    W =  -179.868 deg,    P =   -0.088 deg,    R =   -0.987 deg
};
P[363]{
   GP1:
    UF : 0, UT : 6,      CONFIG : 'N U T, 0, 0, 0',
    X =  350011.060  mm,    Y =   38.933  mm,    Z =   -325807.670  mm,
    W =  -179.992 deg,    P =   0.026 deg,    R =   -1.000 deg
};
P[364]{
   GP1:
    UF : 0, UT : 6,      CONFIG : 'N U T, 0, 0, 0',
    X =  350006.343  mm,    Y =   43.364  mm,    Z =   -325807.400  mm,
    W =  -179.999 deg,    P =   0.015 deg,    R =   -1.000 deg
};
P[365]{
   GP1:
    UF : 0, UT : 6,      CONFIG : 'N U T, 0, 0, 0',
    X =  349940.173  mm,    Y =   106.113  mm,    Z =   -325807.458  mm,
    W =  -179.846 deg,    P =   -0.075 deg,    R =   -0.985 deg
};
P[366]{
   GP1:
    UF : 0, UT : 6,      CONFIG : 'N U T, 0, 0, 0',
    X =  350114.721  mm,    Y =   -100.490  mm,    Z =   -325807.810  mm,
    W =  -180.070 deg,    P =   -0.016 deg,    R =   -0.997 deg
};
P[367]{
   GP1:
    UF : 0, UT : 6,      CONFIG : 'N U T, 0, 0, 0',
    X =  350023.392  mm,    Y =   -22.593  mm,    Z =   -325807.668  mm,
    W =  -179.928 deg,    P =   0.086 deg,    R =   -0.994 deg
};
P[368]{
   GP1:
    UF : 0, UT : 6,      CONFIG : 'N U T, 0, 0, 0',
    X =  349970.490  mm,    Y =   8.398  mm,    Z =   -325807.460  mm,
    W =  -180.011 deg,    P =   0.065 deg,    R =   -0.998 deg
};
P[369]{
   GP1:
    UF : 0, UT : 6,      CONFIG : 'N U T, 0, 0, 0',
    X =  349963.107  mm,    Y =   15.166  mm,    Z =   -325807.480  mm,
    W =  -180.007 deg,    P =   0.054 deg,    R =   -0.999 deg
};
P[370]{
   GP1:
    UF : 0, UT : 6,      CONFIG : 'N U T, 0, 0, 0',
    X =  349967.577  mm,    Y =   4.673  mm,    Z =   -325807.453  mm,
    W =  -180.013 deg,    P =   0.068 deg,    R =   -0.998 deg
};
P[371]{
   GP1:
    UF : 0, UT : 6,      CONFIG : 'N U T, 0, 0, 0',
    X =  349899.498  mm,    Y =   72.748  mm,    Z =   -325807.453  mm,
    W =  -179.870 deg,    P =   0.045 deg,    R =   -0.990 deg
};
P[372]{
   GP1:
    UF : 0, UT : 6,      CONFIG : 'N U T, 0, 0, 0',
    X =  349940.962  mm,    Y =   6.715  mm,    Z =   -325807.602  mm,
    W =  -180.025 deg,    P =   0.099 deg,    R =   -0.995 deg
};
P[373]{
   GP1:
    UF : 0, UT : 6,      CONFIG : 'N U T, 0, 0, 0',
    X =  349988.685  mm,    Y =   -47.181  mm,    Z =   -325807.339  mm,
    W =  -179.937 deg,    P =   0.123 deg,    R =   -0.990 deg
};
P[374]{
   GP1:
    UF : 0, UT : 6,      CONFIG : 'N U T, 0, 0, 0',
    X =  349935.723  mm,    Y =   5.743  mm,    Z =   -325807.701  mm,
    W =  -180.019 deg,    P =   0.118 deg,    R =   -0.993 deg
};
P[375]{
   GP1:
    UF : 0, UT : 6,      CONFIG : 'N U T, 0, 0, 0',
    X =  350040.680  mm,    Y =   -104.256  mm,    Z =   -325807.539  mm,
    W =  -179.944 deg,    P =   0.142 deg,    R =   -0.988 deg
};
P[376]{
   GP1:
    UF : 0, UT : 6,      CONFIG : 'N U T, 0, 0, 0',
    X =  349988.847  mm,    Y =   -58.050  mm,    Z =   -325808.015  mm,
    W =  -179.918 deg,    P =   0.146 deg,    R =   -0.986 deg
};
P[377]{
   GP1:
    UF : 0, UT : 6,      CONFIG : 'N U T, 0, 0, 0',
    X =  350008.350  mm,    Y =   -81.087  mm,    Z =   -325807.613  mm,
    W =  -179.907 deg,    P =   0.202 deg,    R =   -0.975 deg
};
P[378]{
   GP1:
    UF : 0, UT : 6,      CONFIG : 'N U T, 0, 0, 0',
    X =  349912.927  mm,    Y =   4.381  mm,    Z =   -325807.326  mm,
    W =  -180.014 deg,    P =   0.201 deg,    R =   -0.979 deg
};
P[379]{
   GP1:
    UF : 0, UT : 6,      CONFIG : 'N U T, 0, 0, 0',
    X =  349880.747  mm,    Y =   35.030  mm,    Z =   -325807.873  mm,
    W =  -179.887 deg,    P =   0.143 deg,    R =   -0.983 deg
};
P[380]{
   GP1:
    UF : 0, UT : 6,      CONFIG : 'N U T, 0, 0, 0',
    X =  349881.008  mm,    Y =   17.753  mm,    Z =   -325807.522  mm,
    W =  -179.929 deg,    P =   0.180 deg,    R =   -0.981 deg
};
P[381]{
   GP1:
    UF : 0, UT : 6,      CONFIG : 'N U T, 0, 0, 0',
    X =  350037.899  mm,    Y =   6.412  mm,    Z =   -325808.221  mm,
    W =  -179.934 deg,    P =   0.055 deg,    R =   -0.996 deg
};
P[382]{
   GP1:
    UF : 0, UT : 6,      CONFIG : 'N U T, 0, 0, 0',
    X =  350031.037  mm,    Y =   12.249  mm,    Z =   -325808.736  mm,
    W =  -179.955 deg,    P =   0.053 deg,    R =   -0.998 deg
};
P[383]{
   GP1:
    UF : 0, UT : 6,      CONFIG : 'N U T, 0, 0, 0',
    X =  349899.914  mm,    Y =   79.737  mm,    Z =   -325808.810  mm,
    W =  -179.855 deg,    P =   0.036 deg,    R =   -0.989 deg
};
P[384]{
   GP1:
    UF : 0, UT : 6,      CONFIG : 'N U T, 0, 0, 0',
    X =  349969.792  mm,    Y =   1.424  mm,    Z =   -325808.974  mm,
    W =  -180.009 deg,    P =   0.069 deg,    R =   -0.998 deg
};
P[385]{
   GP1:
    UF : 0, UT : 6,      CONFIG : 'N U T, 0, 0, 0',
    X =  349960.411  mm,    Y =   10.805  mm,    Z =   -325808.974  mm,
    W =  -180.014 deg,    P =   0.066 deg,    R =   -0.998 deg
};
P[386]{
   GP1:
    UF : 0, UT : 6,      CONFIG : 'N U T, 0, 0, 0',
    X =  349963.050  mm,    Y =   0.566  mm,    Z =   -325808.599  mm,
    W =  -180.017 deg,    P =   0.081 deg,    R =   -0.997 deg
};
P[387]{
   GP1:
    UF : 0, UT : 6,      CONFIG : 'N U T, 0, 0, 0',
    X =  349955.646  mm,    Y =   7.674  mm,    Z =   -325809.075  mm,
    W =  -180.018 deg,    P =   0.078 deg,    R =   -0.997 deg
};
P[388]{
   GP1:
    UF : 0, UT : 6,      CONFIG : 'N U T, 0, 0, 0',
    X =  349892.240  mm,    Y =   70.955  mm,    Z =   -325808.835  mm,
    W =  -179.851 deg,    P =   0.070 deg,    R =   -0.986 deg
};
P[389]{
   GP1:
    UF : 0, UT : 6,      CONFIG : 'N U T, 0, 0, 0',
    X =  349890.827  mm,    Y =   57.371  mm,    Z =   -325808.189  mm,
    W =  -179.868 deg,    P =   0.084 deg,    R =   -0.988 deg
};
P[390]{
   GP1:
    UF : 0, UT : 6,      CONFIG : 'N U T, 0, 0, 0',
    X =  349904.306  mm,    Y =   0.938  mm,    Z =   -325808.338  mm,
    W =  -180.017 deg,    P =   0.214 deg,    R =   -0.977 deg
};
P[391]{
   GP1:
    UF : 0, UT : 6,      CONFIG : 'N U T, 0, 0, 0',
    X =  349895.241  mm,    Y =   5.574  mm,    Z =   -325808.287  mm,
    W =  -180.000 deg,    P =   0.196 deg,    R =   -0.981 deg
};
P[392]{
   GP1:
    UF : 0, UT : 6,      CONFIG : 'N U T, 0, 0, 0',
    X =  350127.266  mm,    Y =   -37.191  mm,    Z =   -325809.968  mm,
    W =  -180.039 deg,    P =   -0.112 deg,    R =   -0.993 deg
};
P[393]{
   GP1:
    UF : 0, UT : 6,      CONFIG : 'N U T, 0, 0, 0',
    X =  349998.625  mm,    Y =   66.854  mm,    Z =   -325809.775  mm,
    W =  -180.004 deg,    P =   -0.072 deg,    R =   -0.997 deg
};
P[394]{
   GP1:
    UF : 0, UT : 6,      CONFIG : 'N U T, 0, 0, 0',
    X =  350025.040  mm,    Y =   19.677  mm,    Z =   -325809.276  mm,
    W =  -179.962 deg,    P =   0.065 deg,    R =   -0.997 deg
};
P[395]{
   GP1:
    UF : 0, UT : 6,      CONFIG : 'N U T, 0, 0, 0',
    X =  349931.313  mm,    Y =   110.110  mm,    Z =   -325809.292  mm,
    W =  -179.819 deg,    P =   -0.074 deg,    R =   -0.981 deg
};
P[396]{
   GP1:
    UF : 0, UT : 6,      CONFIG : 'N U T, 0, 0, 0',
    X =  349924.018  mm,    Y =   108.625  mm,    Z =   -325809.284  mm,
    W =  -179.816 deg,    P =   -0.057 deg,    R =   -0.981 deg
};
P[397]{
   GP1:
    UF : 0, UT : 6,      CONFIG : 'N U T, 0, 0, 0',
    X =  350035.241  mm,    Y =   -29.808  mm,    Z =   -325809.701  mm,
    W =  -179.920 deg,    P =   0.069 deg,    R =   -0.994 deg
};
P[398]{
   GP1:
    UF : 0, UT : 6,      CONFIG : 'N U T, 0, 0, 0',
    X =  349908.694  mm,    Y =   94.566  mm,    Z =   -325809.383  mm,
    W =  -179.840 deg,    P =   0.012 deg,    R =   -0.987 deg
};
P[399]{
   GP1:
    UF : 0, UT : 6,      CONFIG : 'N U T, 0, 0, 0',
    X =  350112.602  mm,    Y =   -111.159  mm,    Z =   -325810.070  mm,
    W =  -180.076 deg,    P =   -0.007 deg,    R =   -0.997 deg
};
P[400]{
   GP1:
    UF : 0, UT : 6,      CONFIG : 'N U T, 0, 0, 0',
    X =  350036.736  mm,    Y =   -53.058  mm,    Z =   -325809.103  mm,
    W =  -179.927 deg,    P =   0.076 deg,    R =   -0.994 deg
};
P[401]{
   GP1:
    UF : 0, UT : 6,      CONFIG : 'N U T, 0, 0, 0',
    X =  349893.364  mm,    Y =   76.907  mm,    Z =   -325809.706  mm,
    W =  -179.845 deg,    P =   0.053 deg,    R =   -0.986 deg
};
P[402]{
   GP1:
    UF : 0, UT : 6,      CONFIG : 'N U T, 0, 0, 0',
    X =  349997.088  mm,    Y =   -37.551  mm,    Z =   -325809.501  mm,
    W =  -179.936 deg,    P =   0.119 deg,    R =   -0.991 deg
};
P[403]{
   GP1:
    UF : 0, UT : 6,      CONFIG : 'N U T, 0, 0, 0',
    X =  349967.622  mm,    Y =   -7.327  mm,    Z =   -325809.623  mm,
    W =  -180.014 deg,    P =   0.082 deg,    R =   -0.997 deg
};
P[404]{
   GP1:
    UF : 0, UT : 6,      CONFIG : 'N U T, 0, 0, 0',
    X =  349990.888  mm,    Y =   -41.278  mm,    Z =   -325809.201  mm,
    W =  -179.938 deg,    P =   0.119 deg,    R =   -0.991 deg
};
P[405]{
   GP1:
    UF : 0, UT : 6,      CONFIG : 'N U T, 0, 0, 0',
    X =  349961.948  mm,    Y =   -13.770  mm,    Z =   -325809.419  mm,
    W =  -180.014 deg,    P =   0.096 deg,    R =   -0.995 deg
};
P[406]{
   GP1:
    UF : 0, UT : 6,      CONFIG : 'N U T, 0, 0, 0',
    X =  349954.785  mm,    Y =   -6.599  mm,    Z =   -325809.589  mm,
    W =  -180.024 deg,    P =   0.096 deg,    R =   -0.995 deg
};
P[407]{
   GP1:
    UF : 0, UT : 6,      CONFIG : 'N U T, 0, 0, 0',
    X =  349947.731  mm,    Y =   0.463  mm,    Z =   -325809.430  mm,
    W =  -180.027 deg,    P =   0.099 deg,    R =   -0.995 deg
};
P[408]{
   GP1:
    UF : 0, UT : 6,      CONFIG : 'N U T, 0, 0, 0',
    X =  349968.821  mm,    Y =   -21.469  mm,    Z =   -325809.248  mm,
    W =  -180.002 deg,    P =   0.095 deg,    R =   -0.995 deg
};
P[409]{
   GP1:
    UF : 0, UT : 6,      CONFIG : 'N U T, 0, 0, 0',
    X =  349982.592  mm,    Y =   -50.508  mm,    Z =   -325809.611  mm,
    W =  -179.939 deg,    P =   0.124 deg,    R =   -0.990 deg
};
P[410]{
   GP1:
    UF : 0, UT : 6,      CONFIG : 'N U T, 0, 0, 0',
    X =  349925.706  mm,    Y =   6.623  mm,    Z =   -325809.710  mm,
    W =  -180.017 deg,    P =   0.162 deg,    R =   -0.987 deg
};
P[411]{
   GP1:
    UF : 0, UT : 6,      CONFIG : 'N U T, 0, 0, 0',
    X =  349883.333  mm,    Y =   47.596  mm,    Z =   -325809.121  mm,
    W =  -179.870 deg,    P =   0.113 deg,    R =   -0.985 deg
};
P[412]{
   GP1:
    UF : 0, UT : 6,      CONFIG : 'N U T, 0, 0, 0',
    X =  349877.008  mm,    Y =   25.482  mm,    Z =   -325809.518  mm,
    W =  -179.900 deg,    P =   0.170 deg,    R =   -0.980 deg
};
P[413]{
   GP1:
    UF : 0, UT : 6,      CONFIG : 'N U T, 0, 0, 0',
    X =  349943.194  mm,    Y =   110.230  mm,    Z =   -325810.909  mm,
    W =  -179.838 deg,    P =   -0.099 deg,    R =   -0.982 deg
};
P[414]{
   GP1:
    UF : 0, UT : 6,      CONFIG : 'N U T, 0, 0, 0',
    X =  349916.628  mm,    Y =   106.664  mm,    Z =   -325810.157  mm,
    W =  -179.808 deg,    P =   -0.043 deg,    R =   -0.980 deg
};
P[415]{
   GP1:
    UF : 0, UT : 6,      CONFIG : 'N U T, 0, 0, 0',
    X =  350046.985  mm,    Y =   -40.296  mm,    Z =   -325810.361  mm,
    W =  -179.931 deg,    P =   0.056 deg,    R =   -0.996 deg
};
P[416]{
   GP1:
    UF : 0, UT : 6,      CONFIG : 'N U T, 0, 0, 0',
    X =  350048.682  mm,    Y =   -49.201  mm,    Z =   -325810.618  mm,
    W =  -179.940 deg,    P =   0.048 deg,    R =   -0.997 deg
};
P[417]{
   GP1:
    UF : 0, UT : 6,      CONFIG : 'N U T, 0, 0, 0',
    X =  349902.564  mm,    Y =   90.416  mm,    Z =   -325810.530  mm,
    W =  -179.844 deg,    P =   0.024 deg,    R =   -0.988 deg
};
P[418]{
   GP1:
    UF : 0, UT : 6,      CONFIG : 'N U T, 0, 0, 0',
    X =  350042.206  mm,    Y =   -52.143  mm,    Z =   -325810.195  mm,
    W =  -179.931 deg,    P =   0.066 deg,    R =   -0.995 deg
};
P[419]{
   GP1:
    UF : 0, UT : 6,      CONFIG : 'N U T, 0, 0, 0',
    X =  350020.588  mm,    Y =   -39.833  mm,    Z =   -325810.918  mm,
    W =  -179.917 deg,    P =   0.103 deg,    R =   -0.991 deg
};
P[420]{
   GP1:
    UF : 0, UT : 6,      CONFIG : 'N U T, 0, 0, 0',
    X =  349974.762  mm,    Y =   -16.075  mm,    Z =   -325810.934  mm,
    W =  -179.998 deg,    P =   0.086 deg,    R =   -0.996 deg
};
P[421]{
   GP1:
    UF : 0, UT : 6,      CONFIG : 'N U T, 0, 0, 0',
    X =  350070.714  mm,    Y =   -116.108  mm,    Z =   -325810.974  mm,
    W =  -180.020 deg,    P =   0.072 deg,    R =   -0.997 deg
};
P[422]{
   GP1:
    UF : 0, UT : 6,      CONFIG : 'N U T, 0, 0, 0',
    X =  350053.034  mm,    Y =   -109.848  mm,    Z =   -325811.020  mm,
    W =  -179.966 deg,    P =   0.129 deg,    R =   -0.991 deg
};
P[423]{
   GP1:
    UF : 0, UT : 6,      CONFIG : 'N U T, 0, 0, 0',
    X =  349937.383  mm,    Y =   -4.303  mm,    Z =   -325810.853  mm,
    W =  -180.028 deg,    P =   0.140 deg,    R =   -0.990 deg
};
P[424]{
   GP1:
    UF : 0, UT : 6,      CONFIG : 'N U T, 0, 0, 0',
    X =  349933.483  mm,    Y =   0.146  mm,    Z =   -325810.589  mm,
    W =  -180.030 deg,    P =   0.148 deg,    R =   -0.989 deg
};
P[425]{
   GP1:
    UF : 0, UT : 6,      CONFIG : 'N U T, 0, 0, 0',
    X =  349977.261  mm,    Y =   -46.188  mm,    Z =   -325811.005  mm,
    W =  -179.958 deg,    P =   0.122 deg,    R =   -0.992 deg
};
P[426]{
   GP1:
    UF : 0, UT : 6,      CONFIG : 'N U T, 0, 0, 0',
    X =  350118.388  mm,    Y =   -26.806  mm,    Z =   -325811.289  mm,
    W =  -180.003 deg,    P =   -0.126 deg,    R =   -0.992 deg
};
P[427]{
   GP1:
    UF : 0, UT : 6,      CONFIG : 'N U T, 0, 0, 0',
    X =  349986.291  mm,    Y =   86.503  mm,    Z =   -325811.555  mm,
    W =  -179.963 deg,    P =   -0.132 deg,    R =   -0.991 deg
};
P[428]{
   GP1:
    UF : 0, UT : 6,      CONFIG : 'N U T, 0, 0, 0',
    X =  349909.909  mm,    Y =   103.063  mm,    Z =   -325811.361  mm,
    W =  -179.800 deg,    P =   -0.022 deg,    R =   -0.979 deg
};
P[429]{
   GP1:
    UF : 0, UT : 6,      CONFIG : 'N U T, 0, 0, 0',
    X =  350041.301  mm,    Y =   -33.777  mm,    Z =   -325811.234  mm,
    W =  -179.922 deg,    P =   0.066 deg,    R =   -0.995 deg
};
P[430]{
   GP1:
    UF : 0, UT : 6,      CONFIG : 'N U T, 0, 0, 0',
    X =  350027.960  mm,    Y =   -45.698  mm,    Z =   -325811.428  mm,
    W =  -179.918 deg,    P =   0.093 deg,    R =   -0.992 deg
};
P[431]{
   GP1:
    UF : 0, UT : 6,      CONFIG : 'N U T, 0, 0, 0',
    X =  349978.036  mm,    Y =   3.753  mm,    Z =   -325811.594  mm,
    W =  -180.006 deg,    P =   0.066 deg,    R =   -0.998 deg
};
P[432]{
   GP1:
    UF : 0, UT : 6,      CONFIG : 'N U T, 0, 0, 0',
    X =  350007.106  mm,    Y =   -36.363  mm,    Z =   -325811.134  mm,
    W =  -179.928 deg,    P =   0.119 deg,    R =   -0.990 deg
};
P[433]{
   GP1:
    UF : 0, UT : 6,      CONFIG : 'N U T, 0, 0, 0',
    X =  349886.573  mm,    Y =   74.501  mm,    Z =   -325811.653  mm,
    W =  -179.836 deg,    P =   0.075 deg,    R =   -0.984 deg
};
P[434]{
   GP1:
    UF : 0, UT : 6,      CONFIG : 'N U T, 0, 0, 0',
    X =  349981.705  mm,    Y =   -22.213  mm,    Z =   -325811.872  mm,
    W =  -179.977 deg,    P =   0.093 deg,    R =   -0.995 deg
};
P[435]{
   GP1:
    UF : 0, UT : 6,      CONFIG : 'N U T, 0, 0, 0',
    X =  350061.528  mm,    Y =   -112.897  mm,    Z =   -325811.804  mm,
    W =  -179.998 deg,    P =   0.098 deg,    R =   -0.995 deg
};
P[436]{
   GP1:
    UF : 0, UT : 6,      CONFIG : 'N U T, 0, 0, 0',
    X =  349883.143  mm,    Y =   53.449  mm,    Z =   -325811.656  mm,
    W =  -179.861 deg,    P =   0.105 deg,    R =   -0.985 deg
};
P[437]{
   GP1:
    UF : 0, UT : 6,      CONFIG : 'N U T, 0, 0, 0',
    X =  349876.434  mm,    Y =   41.672  mm,    Z =   -325811.979  mm,
    W =  -179.866 deg,    P =   0.136 deg,    R =   -0.982 deg
};
P[438]{
   GP1:
    UF : 0, UT : 6,      CONFIG : 'N U T, 0, 0, 0',
    X =  349994.317  mm,    Y =   79.652  mm,    Z =   -325812.623  mm,
    W =  -180.000 deg,    P =   -0.133 deg,    R =   -0.991 deg
};
P[439]{
   GP1:
    UF : 0, UT : 6,      CONFIG : 'N U T, 0, 0, 0',
    X =  349962.978  mm,    Y =   103.104  mm,    Z =   -325812.379  mm,
    W =  -179.878 deg,    P =   -0.122 deg,    R =   -0.985 deg
};
P[440]{
   GP1:
    UF : 0, UT : 6,      CONFIG : 'N U T, 0, 0, 0',
    X =  349955.617  mm,    Y =   106.322  mm,    Z =   -325812.918  mm,
    W =  -179.862 deg,    P =   -0.115 deg,    R =   -0.984 deg
};
P[441]{
   GP1:
    UF : 0, UT : 6,      CONFIG : 'N U T, 0, 0, 0',
    X =  349925.653  mm,    Y =   114.621  mm,    Z =   -325812.738  mm,
    W =  -179.793 deg,    P =   -0.073 deg,    R =   -0.976 deg
};
P[442]{
   GP1:
    UF : 0, UT : 6,      CONFIG : 'N U T, 0, 0, 0',
    X =  349918.722  mm,    Y =   112.624  mm,    Z =   -325812.953  mm,
    W =  -179.788 deg,    P =   -0.059 deg,    R =   -0.975 deg
};
P[443]{
   GP1:
    UF : 0, UT : 6,      CONFIG : 'N U T, 0, 0, 0',
    X =  350118.233  mm,    Y =   -107.293  mm,    Z =   -325812.162  mm,
    W =  -180.077 deg,    P =   -0.014 deg,    R =   -0.997 deg
};
P[444]{
   GP1:
    UF : 0, UT : 6,      CONFIG : 'N U T, 0, 0, 0',
    X =  349902.340  mm,    Y =   96.510  mm,    Z =   -325812.831  mm,
    W =  -179.812 deg,    P =   0.009 deg,    R =   -0.982 deg
};
P[445]{
   GP1:
    UF : 0, UT : 6,      CONFIG : 'N U T, 0, 0, 0',
    X =  349989.518  mm,    Y =   -0.589  mm,    Z =   -325812.508  mm,
    W =  -179.989 deg,    P =   0.077 deg,    R =   -0.997 deg
};
P[446]{
   GP1:
    UF : 0, UT : 6,      CONFIG : 'N U T, 0, 0, 0',
    X =  349893.617  mm,    Y =   86.532  mm,    Z =   -325812.256  mm,
    W =  -179.827 deg,    P =   0.042 deg,    R =   -0.984 deg
};
P[447]{
   GP1:
    UF : 0, UT : 6,      CONFIG : 'N U T, 0, 0, 0',
    X =  350013.377  mm,    Y =   -35.453  mm,    Z =   -325812.611  mm,
    W =  -179.923 deg,    P =   0.112 deg,    R =   -0.991 deg
};
P[448]{
   GP1:
    UF : 0, UT : 6,      CONFIG : 'N U T, 0, 0, 0',
    X =  349992.449  mm,    Y =   -32.712  mm,    Z =   -325812.157  mm,
    W =  -179.946 deg,    P =   0.109 deg,    R =   -0.993 deg
};
P[449]{
   GP1:
    UF : 0, UT : 6,      CONFIG : 'N U T, 0, 0, 0',
    X =  349977.635  mm,    Y =   -27.227  mm,    Z =   -325812.412  mm,
    W =  -179.980 deg,    P =   0.093 deg,    R =   -0.995 deg
};
P[450]{
   GP1:
    UF : 0, UT : 6,      CONFIG : 'N U T, 0, 0, 0',
    X =  349885.635  mm,    Y =   64.934  mm,    Z =   -325812.448  mm,
    W =  -179.848 deg,    P =   0.084 deg,    R =   -0.985 deg
};
P[451]{
   GP1:
    UF : 0, UT : 6,      CONFIG : 'N U T, 0, 0, 0',
    X =  349976.448  mm,    Y =   -40.844  mm,    Z =   -325812.804  mm,
    W =  -179.966 deg,    P =   0.113 deg,    R =   -0.993 deg
};
P[452]{
   GP1:
    UF : 0, UT : 6,      CONFIG : 'N U T, 0, 0, 0',
    X =  349962.663  mm,    Y =   -27.831  mm,    Z =   -325812.776  mm,
    W =  -180.005 deg,    P =   0.104 deg,    R =   -0.995 deg
};
P[453]{
   GP1:
    UF : 0, UT : 6,      CONFIG : 'N U T, 0, 0, 0',
    X =  349941.002  mm,    Y =   -6.810  mm,    Z =   -325812.233  mm,
    W =  -180.034 deg,    P =   0.138 deg,    R =   -0.990 deg
};
P[454]{
   GP1:
    UF : 0, UT : 6,      CONFIG : 'N U T, 0, 0, 0',
    X =  349933.325  mm,    Y =   -1.832  mm,    Z =   -325812.583  mm,
    W =  -180.030 deg,    P =   0.159 deg,    R =   -0.987 deg
};
P[455]{
   GP1:
    UF : 0, UT : 6,      CONFIG : 'N U T, 0, 0, 0',
    X =  349992.342  mm,    Y =   -67.432  mm,    Z =   -325812.668  mm,
    W =  -179.913 deg,    P =   0.186 deg,    R =   -0.979 deg
};
P[456]{
   GP1:
    UF : 0, UT : 6,      CONFIG : 'N U T, 0, 0, 0',
    X =  349985.798  mm,    Y =   -61.200  mm,    Z =   -325813.073  mm,
    W =  -179.922 deg,    P =   0.169 deg,    R =   -0.983 deg
};
P[457]{
   GP1:
    UF : 0, UT : 6,      CONFIG : 'N U T, 0, 0, 0',
    X =  349917.806  mm,    Y =   1.201  mm,    Z =   -325812.904  mm,
    W =  -180.019 deg,    P =   0.202 deg,    R =   -0.979 deg
};
P[458]{
   GP1:
    UF : 0, UT : 6,      CONFIG : 'N U T, 0, 0, 0',
    X =  349911.007  mm,    Y =   110.214  mm,    Z =   -325813.201  mm,
    W =  -179.783 deg,    P =   -0.041 deg,    R =   -0.975 deg
};
P[459]{
   GP1:
    UF : 0, UT : 6,      CONFIG : 'N U T, 0, 0, 0',
    X =  350030.009  mm,    Y =   -30.484  mm,    Z =   -325813.679  mm,
    W =  -179.916 deg,    P =   0.081 deg,    R =   -0.993 deg
};
P[460]{
   GP1:
    UF : 0, UT : 6,      CONFIG : 'N U T, 0, 0, 0',
    X =  350021.989  mm,    Y =   -24.517  mm,    Z =   -325813.975  mm,
    W =  -179.927 deg,    P =   0.087 deg,    R =   -0.994 deg
};
P[461]{
   GP1:
    UF : 0, UT : 6,      CONFIG : 'N U T, 0, 0, 0',
    X =  349995.477  mm,    Y =   -11.133  mm,    Z =   -325813.887  mm,
    W =  -179.971 deg,    P =   0.093 deg,    R =   -0.995 deg
};
P[462]{
   GP1:
    UF : 0, UT : 6,      CONFIG : 'N U T, 0, 0, 0',
    X =  349973.099  mm,    Y =   -3.670  mm,    Z =   -325813.529  mm,
    W =  -180.010 deg,    P =   0.079 deg,    R =   -0.997 deg
};
P[463]{
   GP1:
    UF : 0, UT : 6,      CONFIG : 'N U T, 0, 0, 0',
    X =  349886.168  mm,    Y =   80.682  mm,    Z =   -325813.222  mm,
    W =  -179.817 deg,    P =   0.073 deg,    R =   -0.980 deg
};
P[464]{
   GP1:
    UF : 0, UT : 6,      CONFIG : 'N U T, 0, 0, 0',
    X =  349984.539  mm,    Y =   -35.402  mm,    Z =   -325813.345  mm,
    W =  -179.960 deg,    P =   0.109 deg,    R =   -0.993 deg
};
P[465]{
   GP1:
    UF : 0, UT : 6,      CONFIG : 'N U T, 0, 0, 0',
    X =  349948.187  mm,    Y =   -13.024  mm,    Z =   -325813.445  mm,
    W =  -180.030 deg,    P =   0.123 deg,    R =   -0.992 deg
};
P[466]{
   GP1:
    UF : 0, UT : 6,      CONFIG : 'N U T, 0, 0, 0',
    X =  349927.051  mm,    Y =   1.453  mm,    Z =   -325813.706  mm,
    W =  -180.019 deg,    P =   0.165 deg,    R =   -0.986 deg
};
P[467]{
   GP1:
    UF : 0, UT : 6,      CONFIG : 'N U T, 0, 0, 0',
    X =  350000.353  mm,    Y =   -74.486  mm,    Z =   -325813.243  mm,
    W =  -179.905 deg,    P =   0.193 deg,    R =   -0.977 deg
};
P[468]{
   GP1:
    UF : 0, UT : 6,      CONFIG : 'N U T, 0, 0, 0',
    X =  349974.470  mm,    Y =   -49.110  mm,    Z =   -325813.757  mm,
    W =  -179.960 deg,    P =   0.137 deg,    R =   -0.990 deg
};
P[469]{
   GP1:
    UF : 0, UT : 6,      CONFIG : 'N U T, 0, 0, 0',
    X =  349978.978  mm,    Y =   -54.136  mm,    Z =   -325813.386  mm,
    W =  -179.941 deg,    P =   0.141 deg,    R =   -0.988 deg
};
P[470]{
   GP1:
    UF : 0, UT : 6,      CONFIG : 'N U T, 0, 0, 0',
    X =  349874.138  mm,    Y =   26.910  mm,    Z =   -325814.010  mm,
    W =  -179.901 deg,    P =   0.168 deg,    R =   -0.981 deg
};
P[471]{
   GP1:
    UF : 0, UT : 6,      CONFIG : 'N U T, 0, 0, 0',
    X =  349884.733  mm,    Y =   6.960  mm,    Z =   -325813.874  mm,
    W =  -179.967 deg,    P =   0.194 deg,    R =   -0.980 deg
};
P[472]{
   GP1:
    UF : 0, UT : 6,      CONFIG : 'N U T, 0, 0, 0',
    X =  350054.698  mm,    Y =   7.474  mm,    Z =   -325814.134  mm,
    W =  -179.916 deg,    P =   0.004 deg,    R =   -0.996 deg
};
P[473]{
   GP1:
    UF : 0, UT : 6,      CONFIG : 'N U T, 0, 0, 0',
    X =  350015.301  mm,    Y =   45.184  mm,    Z =   -325815.051  mm,
    W =  -179.994 deg,    P =   -0.000 deg,    R =   -1.000 deg
};
P[474]{
   GP1:
    UF : 0, UT : 6,      CONFIG : 'N U T, 0, 0, 0',
    X =  349946.689  mm,    Y =   113.280  mm,    Z =   -325814.253  mm,
    W =  -179.841 deg,    P =   -0.116 deg,    R =   -0.980 deg
};
P[475]{
   GP1:
    UF : 0, UT : 6,      CONFIG : 'N U T, 0, 0, 0',
    X =  349937.104  mm,    Y =   115.867  mm,    Z =   -325814.477  mm,
    W =  -179.811 deg,    P =   -0.097 deg,    R =   -0.977 deg
};
P[476]{
   GP1:
    UF : 0, UT : 6,      CONFIG : 'N U T, 0, 0, 0',
    X =  349904.159  mm,    Y =   107.002  mm,    Z =   -325814.718  mm,
    W =  -179.774 deg,    P =   -0.027 deg,    R =   -0.974 deg
};
P[477]{
   GP1:
    UF : 0, UT : 6,      CONFIG : 'N U T, 0, 0, 0',
    X =  350016.514  mm,    Y =   -17.123  mm,    Z =   -325814.645  mm,
    W =  -179.934 deg,    P =   0.091 deg,    R =   -0.994 deg
};
P[478]{
   GP1:
    UF : 0, UT : 6,      CONFIG : 'N U T, 0, 0, 0',
    X =  349896.067  mm,    Y =   93.366  mm,    Z =   -325814.128  mm,
    W =  -179.815 deg,    P =   0.019 deg,    R =   -0.982 deg
};
P[479]{
   GP1:
    UF : 0, UT : 6,      CONFIG : 'N U T, 0, 0, 0',
    X =  350001.096  mm,    Y =   -32.006  mm,    Z =   -325814.241  mm,
    W =  -179.934 deg,    P =   0.115 deg,    R =   -0.991 deg
};
P[480]{
   GP1:
    UF : 0, UT : 6,      CONFIG : 'N U T, 0, 0, 0',
    X =  349986.871  mm,    Y =   -18.621  mm,    Z =   -325814.584  mm,
    W =  -179.973 deg,    P =   0.088 deg,    R =   -0.996 deg
};
P[481]{
   GP1:
    UF : 0, UT : 6,      CONFIG : 'N U T, 0, 0, 0',
    X =  349992.651  mm,    Y =   -25.509  mm,    Z =   -325815.036  mm,
    W =  -179.957 deg,    P =   0.100 deg,    R =   -0.994 deg
};
P[482]{
   GP1:
    UF : 0, UT : 6,      CONFIG : 'N U T, 0, 0, 0',
    X =  349987.276  mm,    Y =   -29.903  mm,    Z =   -325814.556  mm,
    W =  -179.955 deg,    P =   0.100 deg,    R =   -0.994 deg
};
P[483]{
   GP1:
    UF : 0, UT : 6,      CONFIG : 'N U T, 0, 0, 0',
    X =  349882.026  mm,    Y =   70.349  mm,    Z =   -325814.600  mm,
    W =  -179.832 deg,    P =   0.083 deg,    R =   -0.982 deg
};
P[484]{
   GP1:
    UF : 0, UT : 6,      CONFIG : 'N U T, 0, 0, 0',
    X =  350049.739  mm,    Y =   -108.172  mm,    Z =   -325814.871  mm,
    W =  -179.956 deg,    P =   0.127 deg,    R =   -0.991 deg
};
P[485]{
   GP1:
    UF : 0, UT : 6,      CONFIG : 'N U T, 0, 0, 0',
    X =  349970.534  mm,    Y =   -34.609  mm,    Z =   -325814.384  mm,
    W =  -179.981 deg,    P =   0.104 deg,    R =   -0.994 deg
};
P[486]{
   GP1:
    UF : 0, UT : 6,      CONFIG : 'N U T, 0, 0, 0',
    X =  349955.464  mm,    Y =   -19.984  mm,    Z =   -325814.126  mm,
    W =  -180.021 deg,    P =   0.108 deg,    R =   -0.994 deg
};
P[487]{
   GP1:
    UF : 0, UT : 6,      CONFIG : 'N U T, 0, 0, 0',
    X =  350023.608  mm,    Y =   -94.104  mm,    Z =   -325814.606  mm,
    W =  -179.919 deg,    P =   0.180 deg,    R =   -0.980 deg
};
P[488]{
   GP1:
    UF : 0, UT : 6,      CONFIG : 'N U T, 0, 0, 0',
    X =  350016.379  mm,    Y =   -87.526  mm,    Z =   -325814.143  mm,
    W =  -179.912 deg,    P =   0.191 deg,    R =   -0.978 deg
};
P[489]{
   GP1:
    UF : 0, UT : 6,      CONFIG : 'N U T, 0, 0, 0',
    X =  349877.436  mm,    Y =   18.500  mm,    Z =   -325815.003  mm,
    W =  -179.923 deg,    P =   0.183 deg,    R =   -0.980 deg
};
P[490]{
   GP1:
    UF : 0, UT : 6,      CONFIG : 'N U T, 0, 0, 0',
    X =  349889.039  mm,    Y =   4.321  mm,    Z =   -325814.461  mm,
    W =  -179.994 deg,    P =   0.202 deg,    R =   -0.979 deg
};
P[491]{
   GP1:
    UF : 0, UT : 6,      CONFIG : 'N U T, 0, 0, 0',
    X =  349881.235  mm,    Y =   12.124  mm,    Z =   -325814.461  mm,
    W =  -179.949 deg,    P =   0.190 deg,    R =   -0.980 deg
};
P[492]{
   GP1:
    UF : 0, UT : 6,      CONFIG : 'N U T, 0, 0, 0',
    X =  350026.477  mm,    Y =   29.343  mm,    Z =   -325815.672  mm,
    W =  -179.975 deg,    P =   0.030 deg,    R =   -0.999 deg
};
P[493]{
   GP1:
    UF : 0, UT : 6,      CONFIG : 'N U T, 0, 0, 0',
    X =  350032.650  mm,    Y =   20.417  mm,    Z =   -325815.575  mm,
    W =  -179.957 deg,    P =   0.052 deg,    R =   -0.998 deg
};
P[494]{
   GP1:
    UF : 0, UT : 6,      CONFIG : 'N U T, 0, 0, 0',
    X =  350046.725  mm,    Y =   -45.221  mm,    Z =   -325815.098  mm,
    W =  -179.933 deg,    P =   0.056 deg,    R =   -0.996 deg
};
P[495]{
   GP1:
    UF : 0, UT : 6,      CONFIG : 'N U T, 0, 0, 0',
    X =  350008.554  mm,    Y =   -12.811  mm,    Z =   -325815.342  mm,
    W =  -179.947 deg,    P =   0.094 deg,    R =   -0.994 deg
};
P[496]{
   GP1:
    UF : 0, UT : 6,      CONFIG : 'N U T, 0, 0, 0',
    X =  350038.655  mm,    Y =   -47.513  mm,    Z =   -325815.980  mm,
    W =  -179.928 deg,    P =   0.065 deg,    R =   -0.995 deg
};
P[497]{
   GP1:
    UF : 0, UT : 6,      CONFIG : 'N U T, 0, 0, 0',
    X =  350025.345  mm,    Y =   -34.600  mm,    Z =   -325815.920  mm,
    W =  -179.915 deg,    P =   0.089 deg,    R =   -0.992 deg
};
P[498]{
   GP1:
    UF : 0, UT : 6,      CONFIG : 'N U T, 0, 0, 0',
    X =  349888.302  mm,    Y =   91.409  mm,    Z =   -325815.122  mm,
    W =  -179.800 deg,    P =   0.040 deg,    R =   -0.979 deg
};
P[499]{
   GP1:
    UF : 0, UT : 6,      CONFIG : 'N U T, 0, 0, 0',
    X =  349978.639  mm,    Y =   -12.187  mm,    Z =   -325815.522  mm,
    W =  -179.996 deg,    P =   0.082 deg,    R =   -0.997 deg
};
P[500]{
   GP1:
    UF : 0, UT : 6,      CONFIG : 'N U T, 0, 0, 0',
    X =  350082.740  mm,    Y =   -118.121  mm,    Z =   -325815.986  mm,
    W =  -180.041 deg,    P =   0.041 deg,    R =   -0.998 deg
};
P[501]{
   GP1:
    UF : 0, UT : 6,      CONFIG : 'N U T, 0, 0, 0',
    X =  350041.453  mm,    Y =   -104.081  mm,    Z =   -325815.441  mm,
    W =  -179.943 deg,    P =   0.141 deg,    R =   -0.988 deg
};
P[502]{
   GP1:
    UF : 0, UT : 6,      CONFIG : 'N U T, 0, 0, 0',
    X =  349878.566  mm,    Y =   58.367  mm,    Z =   -325815.633  mm,
    W =  -179.841 deg,    P =   0.103 deg,    R =   -0.982 deg
};
P[503]{
   GP1:
    UF : 0, UT : 6,      CONFIG : 'N U T, 0, 0, 0',
    X =  350032.991  mm,    Y =   -99.537  mm,    Z =   -325816.017  mm,
    W =  -179.937 deg,    P =   0.151 deg,    R =   -0.987 deg
};
P[504]{
   GP1:
    UF : 0, UT : 6,      CONFIG : 'N U T, 0, 0, 0',
    X =  349872.123  mm,    Y =   46.935  mm,    Z =   -325815.370  mm,
    W =  -179.858 deg,    P =   0.130 deg,    R =   -0.981 deg
};
P[505]{
   GP1:
    UF : 0, UT : 6,      CONFIG : 'N U T, 0, 0, 0',
    X =  349896.774  mm,    Y =   2.975  mm,    Z =   -325815.159  mm,
    W =  -180.011 deg,    P =   0.206 deg,    R =   -0.978 deg
};
P[506]{
   GP1:
    UF : 0, UT : 6,      CONFIG : 'N U T, 0, 0, 0',
    X =  350007.468  mm,    Y =   57.084  mm,    Z =   -325816.353  mm,
    W =  -180.012 deg,    P =   -0.037 deg,    R =   -0.999 deg
};
P[507]{
   GP1:
    UF : 0, UT : 6,      CONFIG : 'N U T, 0, 0, 0',
    X =  349941.877  mm,    Y =   117.845  mm,    Z =   -325816.847  mm,
    W =  -179.818 deg,    P =   -0.120 deg,    R =   -0.976 deg
};
P[508]{
   GP1:
    UF : 0, UT : 6,      CONFIG : 'N U T, 0, 0, 0',
    X =  350024.360  mm,    Y =   34.865  mm,    Z =   -325816.374  mm,
    W =  -179.983 deg,    P =   0.016 deg,    R =   -1.000 deg
};
P[509]{
   GP1:
    UF : 0, UT : 6,      CONFIG : 'N U T, 0, 0, 0',
    X =  350029.969  mm,    Y =   25.330  mm,    Z =   -325816.435  mm,
    W =  -179.971 deg,    P =   0.041 deg,    R =   -0.999 deg
};
P[510]{
   GP1:
    UF : 0, UT : 6,      CONFIG : 'N U T, 0, 0, 0',
    X =  349920.868  mm,    Y =   119.250  mm,    Z =   -325817.044  mm,
    W =  -179.771 deg,    P =   -0.082 deg,    R =   -0.970 deg
};
P[511]{
   GP1:
    UF : 0, UT : 6,      CONFIG : 'N U T, 0, 0, 0',
    X =  349904.443  mm,    Y =   113.263  mm,    Z =   -325816.536  mm,
    W =  -179.751 deg,    P =   -0.043 deg,    R =   -0.968 deg
};
P[512]{
   GP1:
    UF : 0, UT : 6,      CONFIG : 'N U T, 0, 0, 0',
    X =  349896.833  mm,    Y =   103.583  mm,    Z =   -325817.086  mm,
    W =  -179.767 deg,    P =   -0.007 deg,    R =   -0.972 deg
};
P[513]{
   GP1:
    UF : 0, UT : 6,      CONFIG : 'N U T, 0, 0, 0',
    X =  349993.416  mm,    Y =   -9.199  mm,    Z =   -325816.849  mm,
    W =  -179.976 deg,    P =   0.086 deg,    R =   -0.996 deg
};
P[514]{
   GP1:
    UF : 0, UT : 6,      CONFIG : 'N U T, 0, 0, 0',
    X =  349879.124  mm,    Y =   74.494  mm,    Z =   -325816.681  mm,
    W =  -179.813 deg,    P =   0.083 deg,    R =   -0.979 deg
};
P[515]{
   GP1:
    UF : 0, UT : 6,      CONFIG : 'N U T, 0, 0, 0',
    X =  349922.578  mm,    Y =   -1.035  mm,    Z =   -325816.890  mm,
    W =  -180.029 deg,    P =   0.193 deg,    R =   -0.981 deg
};
P[516]{
   GP1:
    UF : 0, UT : 6,      CONFIG : 'N U T, 0, 0, 0',
    X =  349870.209  mm,    Y =   52.047  mm,    Z =   -325816.895  mm,
    W =  -179.837 deg,    P =   0.123 deg,    R =   -0.979 deg
};
P[517]{
   GP1:
    UF : 0, UT : 6,      CONFIG : 'N U T, 0, 0, 0',
    X =  349870.954  mm,    Y =   35.756  mm,    Z =   -325816.863  mm,
    W =  -179.868 deg,    P =   0.152 deg,    R =   -0.980 deg
};
P[518]{
   GP1:
    UF : 0, UT : 6,      CONFIG : 'N U T, 0, 0, 0',
    X =  349905.038  mm,    Y =   -0.933  mm,    Z =   -325816.435  mm,
    W =  -180.020 deg,    P =   0.213 deg,    R =   -0.977 deg
};
P[519]{
   GP1:
    UF : 0, UT : 6,      CONFIG : 'N U T, 0, 0, 0',
    X =  350106.817  mm,    Y =   -14.152  mm,    Z =   -325817.111  mm,
    W =  -179.936 deg,    P =   -0.153 deg,    R =   -0.986 deg
};
P[520]{
   GP1:
    UF : 0, UT : 6,      CONFIG : 'N U T, 0, 0, 0',
    X =  349992.919  mm,    Y =   89.525  mm,    Z =   -325817.837  mm,
    W =  -179.965 deg,    P =   -0.167 deg,    R =   -0.985 deg
};
P[521]{
   GP1:
    UF : 0, UT : 6,      CONFIG : 'N U T, 0, 0, 0',
    X =  350125.460  mm,    Y =   -94.135  mm,    Z =   -325817.334  mm,
    W =  -180.091 deg,    P =   -0.034 deg,    R =   -0.995 deg
};
P[522]{
   GP1:
    UF : 0, UT : 6,      CONFIG : 'N U T, 0, 0, 0',
    X =  349911.106  mm,    Y =   117.386  mm,    Z =   -325817.091  mm,
    W =  -179.743 deg,    P =   -0.058 deg,    R =   -0.965 deg
};
P[523]{
   GP1:
    UF : 0, UT : 6,      CONFIG : 'N U T, 0, 0, 0',
    X =  350036.816  mm,    Y =   -32.861  mm,    Z =   -325817.335  mm,
    W =  -179.918 deg,    P =   0.065 deg,    R =   -0.995 deg
};
P[524]{
   GP1:
    UF : 0, UT : 6,      CONFIG : 'N U T, 0, 0, 0',
    X =  349889.431  mm,    Y =   98.027  mm,    Z =   -325817.941  mm,
    W =  -179.768 deg,    P =   0.020 deg,    R =   -0.973 deg
};
P[525]{
   GP1:
    UF : 0, UT : 6,      CONFIG : 'N U T, 0, 0, 0',
    X =  349872.619  mm,    Y =   65.748  mm,    Z =   -325817.820  mm,
    W =  -179.817 deg,    P =   0.100 deg,    R =   -0.978 deg
};
P[526]{
   GP1:
    UF : 0, UT : 6,      CONFIG : 'N U T, 0, 0, 0',
    X =  349970.327  mm,    Y =   -48.351  mm,    Z =   -325817.886  mm,
    W =  -179.965 deg,    P =   0.142 deg,    R =   -0.989 deg
};
P[527]{
   GP1:
    UF : 0, UT : 6,      CONFIG : 'N U T, 0, 0, 0',
    X =  349927.957  mm,    Y =   -5.492  mm,    Z =   -325817.834  mm,
    W =  -180.032 deg,    P =   0.193 deg,    R =   -0.981 deg
};
P[528]{
   GP1:
    UF : 0, UT : 6,      CONFIG : 'N U T, 0, 0, 0',
    X =  349911.939  mm,    Y =   -3.518  mm,    Z =   -325818.007  mm,
    W =  -180.030 deg,    P =   0.223 deg,    R =   -0.974 deg
};
P[529]{
   GP1:
    UF : 0, UT : 6,      CONFIG : 'N U T, 0, 0, 0',
    X =  349988.933  mm,    Y =   96.295  mm,    Z =   -325818.489  mm,
    W =  -179.954 deg,    P =   -0.177 deg,    R =   -0.983 deg
};
P[530]{
   GP1:
    UF : 0, UT : 6,      CONFIG : 'N U T, 0, 0, 0',
    X =  349968.677  mm,    Y =   108.798  mm,    Z =   -325818.289  mm,
    W =  -179.876 deg,    P =   -0.161 deg,    R =   -0.979 deg
};
P[531]{
   GP1:
    UF : 0, UT : 6,      CONFIG : 'N U T, 0, 0, 0',
    X =  350045.395  mm,    Y =   14.486  mm,    Z =   -325818.676  mm,
    W =  -179.936 deg,    P =   0.025 deg,    R =   -0.998 deg
};
P[532]{
   GP1:
    UF : 0, UT : 6,      CONFIG : 'N U T, 0, 0, 0',
    X =  350030.597  mm,    Y =   28.217  mm,    Z =   -325818.511  mm,
    W =  -179.972 deg,    P =   0.027 deg,    R =   -0.999 deg
};
P[533]{
   GP1:
    UF : 0, UT : 6,      CONFIG : 'N U T, 0, 0, 0',
    X =  349927.319  mm,    Y =   121.756  mm,    Z =   -325818.381  mm,
    W =  -179.772 deg,    P =   -0.092 deg,    R =   -0.969 deg
};
P[534]{
   GP1:
    UF : 0, UT : 6,      CONFIG : 'N U T, 0, 0, 0',
    X =  349897.643  mm,    Y =   109.189  mm,    Z =   -325818.395  mm,
    W =  -179.752 deg,    P =   -0.023 deg,    R =   -0.969 deg
};
P[535]{
   GP1:
    UF : 0, UT : 6,      CONFIG : 'N U T, 0, 0, 0',
    X =  350033.508  mm,    Y =   -41.662  mm,    Z =   -325818.369  mm,
    W =  -179.919 deg,    P =   0.077 deg,    R =   -0.994 deg
};
P[536]{
   GP1:
    UF : 0, UT : 6,      CONFIG : 'N U T, 0, 0, 0',
    X =  350017.779  mm,    Y =   -28.740  mm,    Z =   -325818.490  mm,
    W =  -179.923 deg,    P =   0.100 deg,    R =   -0.992 deg
};
P[537]{
   GP1:
    UF : 0, UT : 6,      CONFIG : 'N U T, 0, 0, 0',
    X =  349982.453  mm,    Y =   2.520  mm,    Z =   -325818.363  mm,
    W =  -180.001 deg,    P =   0.068 deg,    R =   -0.998 deg
};
P[538]{
   GP1:
    UF : 0, UT : 6,      CONFIG : 'N U T, 0, 0, 0',
    X =  349881.106  mm,    Y =   87.279  mm,    Z =   -325818.091  mm,
    W =  -179.790 deg,    P =   0.070 deg,    R =   -0.975 deg
};
P[539]{
   GP1:
    UF : 0, UT : 6,      CONFIG : 'N U T, 0, 0, 0',
    X =  349874.095  mm,    Y =   72.046  mm,    Z =   -325818.400  mm,
    W =  -179.810 deg,    P =   0.094 deg,    R =   -0.977 deg
};
P[540]{
   GP1:
    UF : 0, UT : 6,      CONFIG : 'N U T, 0, 0, 0',
    X =  349865.183  mm,    Y =   58.739  mm,    Z =   -325818.929  mm,
    W =  -179.817 deg,    P =   0.122 deg,    R =   -0.975 deg
};
P[541]{
   GP1:
    UF : 0, UT : 6,      CONFIG : 'N U T, 0, 0, 0',
    X =  349964.255  mm,    Y =   -40.892  mm,    Z =   -325818.807  mm,
    W =  -179.989 deg,    P =   0.134 deg,    R =   -0.991 deg
};
P[542]{
   GP1:
    UF : 0, UT : 6,      CONFIG : 'N U T, 0, 0, 0',
    X =  349977.188  mm,    Y =   -55.981  mm,    Z =   -325818.975  mm,
    W =  -179.944 deg,    P =   0.156 deg,    R =   -0.986 deg
};
P[543]{
   GP1:
    UF : 0, UT : 6,      CONFIG : 'N U T, 0, 0, 0',
    X =  349868.598  mm,    Y =   43.230  mm,    Z =   -325818.519  mm,
    W =  -179.860 deg,    P =   0.137 deg,    R =   -0.981 deg
};
P[544]{
   GP1:
    UF : 0, UT : 6,      CONFIG : 'N U T, 0, 0, 0',
    X =  349984.347  mm,    Y =   105.758  mm,    Z =   -325819.770  mm,
    W =  -179.915 deg,    P =   -0.206 deg,    R =   -0.975 deg
};
P[545]{
   GP1:
    UF : 0, UT : 6,      CONFIG : 'N U T, 0, 0, 0',
    X =  350003.542  mm,    Y =   78.508  mm,    Z =   -325819.967  mm,
    W =  -180.010 deg,    P =   -0.147 deg,    R =   -0.989 deg
};
P[546]{
   GP1:
    UF : 0, UT : 6,      CONFIG : 'N U T, 0, 0, 0',
    X =  350142.789  mm,    Y =   -65.394  mm,    Z =   -325819.455  mm,
    W =  -180.135 deg,    P =   -0.108 deg,    R =   -0.985 deg
};
P[547]{
   GP1:
    UF : 0, UT : 6,      CONFIG : 'N U T, 0, 0, 0',
    X =  349959.822  mm,    Y =   112.883  mm,    Z =   -325819.327  mm,
    W =  -179.844 deg,    P =   -0.140 deg,    R =   -0.978 deg
};
P[548]{
   GP1:
    UF : 0, UT : 6,      CONFIG : 'N U T, 0, 0, 0',
    X =  349989.138  mm,    Y =   -0.598  mm,    Z =   -325820.067  mm,
    W =  -179.988 deg,    P =   0.078 deg,    R =   -0.997 deg
};
P[549]{
   GP1:
    UF : 0, UT : 6,      CONFIG : 'N U T, 0, 0, 0',
    X =  350001.848  mm,    Y =   -14.846  mm,    Z =   -325819.699  mm,
    W =  -179.955 deg,    P =   0.094 deg,    R =   -0.995 deg
};
P[550]{
   GP1:
    UF : 0, UT : 6,      CONFIG : 'N U T, 0, 0, 0',
    X =  350004.199  mm,    Y =   -26.278  mm,    Z =   -325820.044  mm,
    W =  -179.932 deg,    P =   0.110 deg,    R =   -0.992 deg
};
P[551]{
   GP1:
    UF : 0, UT : 6,      CONFIG : 'N U T, 0, 0, 0',
    X =  349999.725  mm,    Y =   -22.061  mm,    Z =   -325819.999  mm,
    W =  -179.953 deg,    P =   0.104 deg,    R =   -0.993 deg
};
P[552]{
   GP1:
    UF : 0, UT : 6,      CONFIG : 'N U T, 0, 0, 0',
    X =  349988.520  mm,    Y =   -11.286  mm,    Z =   -325819.169  mm,
    W =  -179.982 deg,    P =   0.088 deg,    R =   -0.996 deg
};
P[553]{
   GP1:
    UF : 0, UT : 6,      CONFIG : 'N U T, 0, 0, 0',
    X =  350072.236  mm,    Y =   -115.037  mm,    Z =   -325819.229  mm,
    W =  -180.020 deg,    P =   0.067 deg,    R =   -0.998 deg
};
P[554]{
   GP1:
    UF : 0, UT : 6,      CONFIG : 'N U T, 0, 0, 0',
    X =  349873.844  mm,    Y =   81.366  mm,    Z =   -325819.759  mm,
    W =  -179.782 deg,    P =   0.079 deg,    R =   -0.973 deg
};
P[555]{
   GP1:
    UF : 0, UT : 6,      CONFIG : 'N U T, 0, 0, 0',
    X =  349867.091  mm,    Y =   70.261  mm,    Z =   -325819.851  mm,
    W =  -179.798 deg,    P =   0.113 deg,    R =   -0.973 deg
};
P[556]{
   GP1:
    UF : 0, UT : 6,      CONFIG : 'N U T, 0, 0, 0',
    X =  350007.933  mm,    Y =   -81.223  mm,    Z =   -325819.839  mm,
    W =  -179.904 deg,    P =   0.204 deg,    R =   -0.974 deg
};
P[557]{
   GP1:
    UF : 0, UT : 6,      CONFIG : 'N U T, 0, 0, 0',
    X =  349943.388  mm,    Y =   -18.978  mm,    Z =   -325819.840  mm,
    W =  -180.037 deg,    P =   0.150 deg,    R =   -0.988 deg
};
P[558]{
   GP1:
    UF : 0, UT : 6,      CONFIG : 'N U T, 0, 0, 0',
    X =  349935.629  mm,    Y =   -11.981  mm,    Z =   -325819.374  mm,
    W =  -180.036 deg,    P =   0.172 deg,    R =   -0.984 deg
};
P[559]{
   GP1:
    UF : 0, UT : 6,      CONFIG : 'N U T, 0, 0, 0',
    X =  349984.430  mm,    Y =   -62.763  mm,    Z =   -325819.579  mm,
    W =  -179.920 deg,    P =   0.172 deg,    R =   -0.982 deg
};
P[560]{
   GP1:
    UF : 0, UT : 6,      CONFIG : 'N U T, 0, 0, 0',
    X =  349915.210  mm,    Y =   123.350  mm,    Z =   -325821.028  mm,
    W =  -179.736 deg,    P =   -0.078 deg,    R =   -0.961 deg
};
P[561]{
   GP1:
    UF : 0, UT : 6,      CONFIG : 'N U T, 0, 0, 0',
    X =  349890.249  mm,    Y =   106.416  mm,    Z =   -325820.923  mm,
    W =  -179.740 deg,    P =   -0.003 deg,    R =   -0.966 deg
};
P[562]{
   GP1:
    UF : 0, UT : 6,      CONFIG : 'N U T, 0, 0, 0',
    X =  349979.608  mm,    Y =   -1.276  mm,    Z =   -325820.644  mm,
    W =  -180.003 deg,    P =   0.071 deg,    R =   -0.997 deg
};
P[563]{
   GP1:
    UF : 0, UT : 6,      CONFIG : 'N U T, 0, 0, 0',
    X =  349881.350  mm,    Y =   93.340  mm,    Z =   -325820.502  mm,
    W =  -179.762 deg,    P =   0.056 deg,    R =   -0.970 deg
};
P[564]{
   GP1:
    UF : 0, UT : 6,      CONFIG : 'N U T, 0, 0, 0',
    X =  350078.820  mm,    Y =   -116.825  mm,    Z =   -325820.371  mm,
    W =  -180.020 deg,    P =   0.040 deg,    R =   -0.999 deg
};
P[565]{
   GP1:
    UF : 0, UT : 6,      CONFIG : 'N U T, 0, 0, 0',
    X =  350023.438  mm,    Y =   -93.753  mm,    Z =   -325820.563  mm,
    W =  -179.915 deg,    P =   0.184 deg,    R =   -0.979 deg
};
P[566]{
   GP1:
    UF : 0, UT : 6,      CONFIG : 'N U T, 0, 0, 0',
    X =  350015.888  mm,    Y =   -87.322  mm,    Z =   -325820.136  mm,
    W =  -179.904 deg,    P =   0.197 deg,    R =   -0.976 deg
};
P[567]{
   GP1:
    UF : 0, UT : 6,      CONFIG : 'N U T, 0, 0, 0',
    X =  349958.032  mm,    Y =   -32.935  mm,    Z =   -325821.067  mm,
    W =  -180.010 deg,    P =   0.126 deg,    R =   -0.992 deg
};
P[568]{
   GP1:
    UF : 0, UT : 6,      CONFIG : 'N U T, 0, 0, 0',
    X =  349992.563  mm,    Y =   -68.707  mm,    Z =   -325820.751  mm,
    W =  -179.910 deg,    P =   0.186 deg,    R =   -0.978 deg
};
P[569]{
   GP1:
    UF : 0, UT : 6,      CONFIG : 'N U T, 0, 0, 0',
    X =  349878.591  mm,    Y =   15.472  mm,    Z =   -325820.539  mm,
    W =  -179.928 deg,    P =   0.186 deg,    R =   -0.980 deg
};
P[570]{
   GP1:
    UF : 0, UT : 6,      CONFIG : 'N U T, 0, 0, 0',
    X =  349984.967  mm,    Y =   107.366  mm,    Z =   -325821.764  mm,
    W =  -179.909 deg,    P =   -0.235 deg,    R =   -0.968 deg
};
P[571]{
   GP1:
    UF : 0, UT : 6,      CONFIG : 'N U T, 0, 0, 0',
    X =  350007.948  mm,    Y =   72.065  mm,    Z =   -325821.866  mm,
    W =  -180.018 deg,    P =   -0.124 deg,    R =   -0.992 deg
};
P[572]{
   GP1:
    UF : 0, UT : 6,      CONFIG : 'N U T, 0, 0, 0',
    X =  350010.431  mm,    Y =   62.031  mm,    Z =   -325821.194  mm,
    W =  -180.021 deg,    P =   -0.073 deg,    R =   -0.997 deg
};
P[573]{
   GP1:
    UF : 0, UT : 6,      CONFIG : 'N U T, 0, 0, 0',
    X =  350058.771  mm,    Y =   12.814  mm,    Z =   -325821.638  mm,
    W =  -179.916 deg,    P =   -0.023 deg,    R =   -0.996 deg
};
P[574]{
   GP1:
    UF : 0, UT : 6,      CONFIG : 'N U T, 0, 0, 0',
    X =  350015.674  mm,    Y =   54.008  mm,    Z =   -325821.139  mm,
    W =  -180.015 deg,    P =   -0.049 deg,    R =   -0.999 deg
};
P[575]{
   GP1:
    UF : 0, UT : 6,      CONFIG : 'N U T, 0, 0, 0',
    X =  349922.199  mm,    Y =   125.253  mm,    Z =   -325821.648  mm,
    W =  -179.741 deg,    P =   -0.094 deg,    R =   -0.961 deg
};
P[576]{
   GP1:
    UF : 0, UT : 6,      CONFIG : 'N U T, 0, 0, 0',
    X =  350129.459  mm,    Y =   -93.472  mm,    Z =   -325821.999  mm,
    W =  -180.093 deg,    P =   -0.039 deg,    R =   -0.995 deg
};
P[577]{
   GP1:
    UF : 0, UT : 6,      CONFIG : 'N U T, 0, 0, 0',
    X =  349899.311  mm,    Y =   119.016  mm,    Z =   -325821.131  mm,
    W =  -179.720 deg,    P =   -0.048 deg,    R =   -0.959 deg
};
P[578]{
   GP1:
    UF : 0, UT : 6,      CONFIG : 'N U T, 0, 0, 0',
    X =  350009.322  mm,    Y =   -25.548  mm,    Z =   -325821.713  mm,
    W =  -179.933 deg,    P =   0.105 deg,    R =   -0.992 deg
};
P[579]{
   GP1:
    UF : 0, UT : 6,      CONFIG : 'N U T, 0, 0, 0',
    X =  350063.834  mm,    Y =   -111.976  mm,    Z =   -325821.775  mm,
    W =  -179.999 deg,    P =   0.079 deg,    R =   -0.997 deg
};
P[580]{
   GP1:
    UF : 0, UT : 6,      CONFIG : 'N U T, 0, 0, 0',
    X =  349866.919  mm,    Y =   76.019  mm,    Z =   -325821.713  mm,
    W =  -179.777 deg,    P =   0.098 deg,    R =   -0.970 deg
};
P[581]{
   GP1:
    UF : 0, UT : 6,      CONFIG : 'N U T, 0, 0, 0',
    X =  350030.741  mm,    Y =   -98.501  mm,    Z =   -325821.364  mm,
    W =  -179.930 deg,    P =   0.163 deg,    R =   -0.984 deg
};
P[582]{
   GP1:
    UF : 0, UT : 6,      CONFIG : 'N U T, 0, 0, 0',
    X =  350000.322  mm,    Y =   -74.763  mm,    Z =   -325821.115  mm,
    W =  -179.905 deg,    P =   0.201 deg,    R =   -0.975 deg
};
P[583]{
   GP1:
    UF : 0, UT : 6,      CONFIG : 'N U T, 0, 0, 0',
    X =  349873.231  mm,    Y =   24.270  mm,    Z =   -325821.823  mm,
    W =  -179.899 deg,    P =   0.170 deg,    R =   -0.980 deg
};
P[584]{
   GP1:
    UF : 0, UT : 6,      CONFIG : 'N U T, 0, 0, 0',
    X =  349891.996  mm,    Y =   0.923  mm,    Z =   -325821.716  mm,
    W =  -180.006 deg,    P =   0.200 deg,    R =   -0.980 deg
};
P[585]{
   GP1:
    UF : 0, UT : 6,      CONFIG : 'N U T, 0, 0, 0',
    X =  349883.415  mm,    Y =   6.574  mm,    Z =   -325821.745  mm,
    W =  -179.970 deg,    P =   0.202 deg,    R =   -0.979 deg
};
P[586]{
   GP1:
    UF : 0, UT : 6,      CONFIG : 'N U T, 0, 0, 0',
    X =  350133.145  mm,    Y =   -23.134  mm,    Z =   -325822.481  mm,
    W =  -180.022 deg,    P =   -0.207 deg,    R =   -0.978 deg
};
P[587]{
   GP1:
    UF : 0, UT : 6,      CONFIG : 'N U T, 0, 0, 0',
    X =  350118.723  mm,    Y =   -15.140  mm,    Z =   -325822.632  mm,
    W =  -179.965 deg,    P =   -0.187 deg,    R =   -0.982 deg
};
P[588]{
   GP1:
    UF : 0, UT : 6,      CONFIG : 'N U T, 0, 0, 0',
    X =  349965.910  mm,    Y =   113.835  mm,    Z =   -325822.249  mm,
    W =  -179.857 deg,    P =   -0.170 deg,    R =   -0.975 deg
};
P[589]{
   GP1:
    UF : 0, UT : 6,      CONFIG : 'N U T, 0, 0, 0',
    X =  350146.028  mm,    Y =   -66.543  mm,    Z =   -325822.633  mm,
    W =  -180.191 deg,    P =   -0.127 deg,    R =   -0.973 deg
};
P[590]{
   GP1:
    UF : 0, UT : 6,      CONFIG : 'N U T, 0, 0, 0',
    X =  349954.770  mm,    Y =   120.032  mm,    Z =   -325822.351  mm,
    W =  -179.828 deg,    P =   -0.158 deg,    R =   -0.972 deg
};
P[591]{
   GP1:
    UF : 0, UT : 6,      CONFIG : 'N U T, 0, 0, 0',
    X =  349944.558  mm,    Y =   124.284  mm,    Z =   -325822.604  mm,
    W =  -179.803 deg,    P =   -0.152 deg,    R =   -0.969 deg
};
P[592]{
   GP1:
    UF : 0, UT : 6,      CONFIG : 'N U T, 0, 0, 0',
    X =  350029.343  mm,    Y =   38.743  mm,    Z =   -325822.811  mm,
    W =  -179.983 deg,    P =   -0.004 deg,    R =   -1.000 deg
};
P[593]{
   GP1:
    UF : 0, UT : 6,      CONFIG : 'N U T, 0, 0, 0',
    X =  350046.324  mm,    Y =   -39.454  mm,    Z =   -325823.061  mm,
    W =  -179.929 deg,    P =   0.055 deg,    R =   -0.996 deg
};
P[594]{
   GP1:
    UF : 0, UT : 6,      CONFIG : 'N U T, 0, 0, 0',
    X =  349892.203  mm,    Y =   113.977  mm,    Z =   -325822.975  mm,
    W =  -179.716 deg,    P =   -0.017 deg,    R =   -0.959 deg
};
P[595]{
   GP1:
    UF : 0, UT : 6,      CONFIG : 'N U T, 0, 0, 0',
    X =  350040.545  mm,    Y =   -35.031  mm,    Z =   -325822.623  mm,
    W =  -179.921 deg,    P =   0.067 deg,    R =   -0.995 deg
};
P[596]{
   GP1:
    UF : 0, UT : 6,      CONFIG : 'N U T, 0, 0, 0',
    X =  350019.051  mm,    Y =   -20.832  mm,    Z =   -325822.606  mm,
    W =  -179.927 deg,    P =   0.087 deg,    R =   -0.994 deg
};
P[597]{
   GP1:
    UF : 0, UT : 6,      CONFIG : 'N U T, 0, 0, 0',
    X =  350011.681  mm,    Y =   -13.462  mm,    Z =   -325822.606  mm,
    W =  -179.942 deg,    P =   0.088 deg,    R =   -0.994 deg
};
P[598]{
   GP1:
    UF : 0, UT : 6,      CONFIG : 'N U T, 0, 0, 0',
    X =  349884.875  mm,    Y =   103.946  mm,    Z =   -325822.614  mm,
    W =  -179.727 deg,    P =   0.017 deg,    R =   -0.962 deg
};
P[599]{
   GP1:
    UF : 0, UT : 6,      CONFIG : 'N U T, 0, 0, 0',
    X =  349984.013  mm,    Y =   -5.433  mm,    Z =   -325822.628  mm,
    W =  -179.995 deg,    P =   0.080 deg,    R =   -0.997 deg
};
P[600]{
   GP1:
    UF : 0, UT : 6,      CONFIG : 'N U T, 0, 0, 0',
    X =  349951.488  mm,    Y =   -25.148  mm,    Z =   -325822.304  mm,
    W =  -180.026 deg,    P =   0.135 deg,    R =   -0.991 deg
};
P[601]{
   GP1:
    UF : 0, UT : 6,      CONFIG : 'N U T, 0, 0, 0',
    X =  349869.824  mm,    Y =   30.744  mm,    Z =   -325822.227  mm,
    W =  -179.884 deg,    P =   0.169 deg,    R =   -0.979 deg
};
P[602]{
   GP1:
    UF : 0, UT : 6,      CONFIG : 'N U T, 0, 0, 0',
    X =  350125.417  mm,    Y =   -16.478  mm,    Z =   -325824.017  mm,
    W =  -180.001 deg,    P =   -0.201 deg,    R =   -0.980 deg
};
P[603]{
   GP1:
    UF : 0, UT : 6,      CONFIG : 'N U T, 0, 0, 0',
    X =  349992.315  mm,    Y =   100.177  mm,    Z =   -325823.403  mm,
    W =  -179.943 deg,    P =   -0.221 deg,    R =   -0.974 deg
};
P[604]{
   GP1:
    UF : 0, UT : 6,      CONFIG : 'N U T, 0, 0, 0',
    X =  350023.081  mm,    Y =   49.692  mm,    Z =   -325824.022  mm,
    W =  -179.995 deg,    P =   -0.027 deg,    R =   -1.000 deg
};
P[605]{
   GP1:
    UF : 0, UT : 6,      CONFIG : 'N U T, 0, 0, 0',
    X =  350050.453  mm,    Y =   17.650  mm,    Z =   -325823.891  mm,
    W =  -179.933 deg,    P =   -0.009 deg,    R =   -0.998 deg
};
P[606]{
   GP1:
    UF : 0, UT : 6,      CONFIG : 'N U T, 0, 0, 0',
    X =  350035.448  mm,    Y =   30.033  mm,    Z =   -325823.224  mm,
    W =  -179.968 deg,    P =   0.012 deg,    R =   -0.999 deg
};
P[607]{
   GP1:
    UF : 0, UT : 6,      CONFIG : 'N U T, 0, 0, 0',
    X =  350042.138  mm,    Y =   22.481  mm,    Z =   -325823.237  mm,
    W =  -179.951 deg,    P =   0.010 deg,    R =   -0.999 deg
};
P[608]{
   GP1:
    UF : 0, UT : 6,      CONFIG : 'N U T, 0, 0, 0',
    X =  349930.627  mm,    Y =   128.181  mm,    Z =   -325823.608  mm,
    W =  -179.753 deg,    P =   -0.130 deg,    R =   -0.960 deg
};
P[609]{
   GP1:
    UF : 0, UT : 6,      CONFIG : 'N U T, 0, 0, 0',
    X =  350016.289  mm,    Y =   -16.237  mm,    Z =   -325823.238  mm,
    W =  -179.935 deg,    P =   0.090 deg,    R =   -0.994 deg
};
P[610]{
   GP1:
    UF : 0, UT : 6,      CONFIG : 'N U T, 0, 0, 0',
    X =  350017.799  mm,    Y =   -22.925  mm,    Z =   -325823.864  mm,
    W =  -179.927 deg,    P =   0.097 deg,    R =   -0.993 deg
};
P[611]{
   GP1:
    UF : 0, UT : 6,      CONFIG : 'N U T, 0, 0, 0',
    X =  349868.910  mm,    Y =   87.096  mm,    Z =   -325823.676  mm,
    W =  -179.744 deg,    P =   0.078 deg,    R =   -0.963 deg
};
P[612]{
   GP1:
    UF : 0, UT : 6,      CONFIG : 'N U T, 0, 0, 0',
    X =  350058.938  mm,    Y =   -110.413  mm,    Z =   -325823.623  mm,
    W =  -179.973 deg,    P =   0.099 deg,    R =   -0.995 deg
};
P[613]{
   GP1:
    UF : 0, UT : 6,      CONFIG : 'N U T, 0, 0, 0',
    X =  349861.262  mm,    Y =   66.016  mm,    Z =   -325823.108  mm,
    W =  -179.794 deg,    P =   0.120 deg,    R =   -0.971 deg
};
P[614]{
   GP1:
    UF : 0, UT : 6,      CONFIG : 'N U T, 0, 0, 0',
    X =  349865.019  mm,    Y =   45.314  mm,    Z =   -325823.669  mm,
    W =  -179.835 deg,    P =   0.142 deg,    R =   -0.976 deg
};
P[615]{
   GP1:
    UF : 0, UT : 6,      CONFIG : 'N U T, 0, 0, 0',
    X =  349915.957  mm,    Y =   -6.201  mm,    Z =   -325823.127  mm,
    W =  -180.032 deg,    P =   0.225 deg,    R =   -0.974 deg
};
P[616]{
   GP1:
    UF : 0, UT : 6,      CONFIG : 'N U T, 0, 0, 0',
    X =  349867.494  mm,    Y =   37.755  mm,    Z =   -325823.299  mm,
    W =  -179.865 deg,    P =   0.155 deg,    R =   -0.979 deg
};
P[617]{
   GP1:
    UF : 0, UT : 6,      CONFIG : 'N U T, 0, 0, 0',
    X =  349906.293  mm,    Y =   -7.963  mm,    Z =   -325823.919  mm,
    W =  -180.037 deg,    P =   0.228 deg,    R =   -0.973 deg
};
P[618]{
   GP1:
    UF : 0, UT : 6,      CONFIG : 'N U T, 0, 0, 0',
    X =  349901.341  mm,    Y =   -4.008  mm,    Z =   -325823.613  mm,
    W =  -180.022 deg,    P =   0.213 deg,    R =   -0.977 deg
};
P[619]{
   GP1:
    UF : 0, UT : 6,      CONFIG : 'N U T, 0, 0, 0',
    X =  350110.906  mm,    Y =   -8.229  mm,    Z =   -325824.106  mm,
    W =  -179.929 deg,    P =   -0.177 deg,    R =   -0.982 deg
};
P[620]{
   GP1:
    UF : 0, UT : 6,      CONFIG : 'N U T, 0, 0, 0',
    X =  349999.503  mm,    Y =   93.684  mm,    Z =   -325825.029  mm,
    W =  -179.977 deg,    P =   -0.215 deg,    R =   -0.976 deg
};
P[621]{
   GP1:
    UF : 0, UT : 6,      CONFIG : 'N U T, 0, 0, 0',
    X =  349974.778  mm,    Y =   114.918  mm,    Z =   -325825.020  mm,
    W =  -179.860 deg,    P =   -0.204 deg,    R =   -0.969 deg
};
P[622]{
   GP1:
    UF : 0, UT : 6,      CONFIG : 'N U T, 0, 0, 0',
    X =  349955.944  mm,    Y =   123.329  mm,    Z =   -325824.975  mm,
    W =  -179.824 deg,    P =   -0.179 deg,    R =   -0.968 deg
};
P[623]{
   GP1:
    UF : 0, UT : 6,      CONFIG : 'N U T, 0, 0, 0',
    X =  350131.724  mm,    Y =   -95.376  mm,    Z =   -325824.978  mm,
    W =  -180.135 deg,    P =   -0.056 deg,    R =   -0.989 deg
};
P[624]{
   GP1:
    UF : 0, UT : 6,      CONFIG : 'N U T, 0, 0, 0',
    X =  349907.698  mm,    Y =   128.251  mm,    Z =   -325825.029  mm,
    W =  -179.706 deg,    P =   -0.079 deg,    R =   -0.953 deg
};
P[625]{
   GP1:
    UF : 0, UT : 6,      CONFIG : 'N U T, 0, 0, 0',
    X =  349900.539  mm,    Y =   125.055  mm,    Z =   -325824.203  mm,
    W =  -179.704 deg,    P =   -0.065 deg,    R =   -0.953 deg
};
P[626]{
   GP1:
    UF : 0, UT : 6,      CONFIG : 'N U T, 0, 0, 0',
    X =  349876.884  mm,    Y =   98.338  mm,    Z =   -325824.990  mm,
    W =  -179.721 deg,    P =   0.046 deg,    R =   -0.959 deg
};
P[627]{
   GP1:
    UF : 0, UT : 6,      CONFIG : 'N U T, 0, 0, 0',
    X =  350052.347  mm,    Y =   -108.073  mm,    Z =   -325824.414  mm,
    W =  -179.957 deg,    P =   0.121 deg,    R =   -0.992 deg
};
P[628]{
   GP1:
    UF : 0, UT : 6,      CONFIG : 'N U T, 0, 0, 0',
    X =  350147.855  mm,    Y =   -58.641  mm,    Z =   -325825.204  mm,
    W =  -180.216 deg,    P =   -0.165 deg,    R =   -0.962 deg
};
P[629]{
   GP1:
    UF : 0, UT : 6,      CONFIG : 'N U T, 0, 0, 0',
    X =  350014.548  mm,    Y =   64.004  mm,    Z =   -325826.002  mm,
    W =  -180.026 deg,    P =   -0.101 deg,    R =   -0.995 deg
};
P[630]{
   GP1:
    UF : 0, UT : 6,      CONFIG : 'N U T, 0, 0, 0',
    X =  349936.249  mm,    Y =   129.830  mm,    Z =   -325825.405  mm,
    W =  -179.755 deg,    P =   -0.145 deg,    R =   -0.959 deg
};
P[631]{
   GP1:
    UF : 0, UT : 6,      CONFIG : 'N U T, 0, 0, 0',
    X =  350008.500  mm,    Y =   -14.114  mm,    Z =   -325825.708  mm,
    W =  -179.947 deg,    P =   0.095 deg,    R =   -0.994 deg
};
P[632]{
   GP1:
    UF : 0, UT : 6,      CONFIG : 'N U T, 0, 0, 0',
    X =  349883.725  mm,    Y =   109.512  mm,    Z =   -325825.366  mm,
    W =  -179.695 deg,    P =   0.007 deg,    R =   -0.952 deg
};
P[633]{
   GP1:
    UF : 0, UT : 6,      CONFIG : 'N U T, 0, 0, 0',
    X =  349987.818  mm,    Y =   -0.891  mm,    Z =   -325825.719  mm,
    W =  -179.992 deg,    P =   0.076 deg,    R =   -0.997 deg
};
P[634]{
   GP1:
    UF : 0, UT : 6,      CONFIG : 'N U T, 0, 0, 0',
    X =  350043.094  mm,    Y =   -103.717  mm,    Z =   -325825.153  mm,
    W =  -179.943 deg,    P =   0.138 deg,    R =   -0.989 deg
};
P[635]{
   GP1:
    UF : 0, UT : 6,      CONFIG : 'N U T, 0, 0, 0',
    X =  349923.553  mm,    Y =   -8.254  mm,    Z =   -325825.947  mm,
    W =  -180.038 deg,    P =   0.211 deg,    R =   -0.977 deg
};
P[636]{
   GP1:
    UF : 0, UT : 6,      CONFIG : 'N U T, 0, 0, 0',
    X =  349861.193  mm,    Y =   53.280  mm,    Z =   -325825.738  mm,
    W =  -179.815 deg,    P =   0.139 deg,    R =   -0.973 deg
};
P[637]{
   GP1:
    UF : 0, UT : 6,      CONFIG : 'N U T, 0, 0, 0',
    X =  349958.979  mm,    Y =   -45.663  mm,    Z =   -325825.647  mm,
    W =  -179.997 deg,    P =   0.153 deg,    R =   -0.988 deg
};
P[638]{
   GP1:
    UF : 0, UT : 6,      CONFIG : 'N U T, 0, 0, 0',
    X =  350146.694  mm,    Y =   -46.581  mm,    Z =   -325826.203  mm,
    W =  -180.190 deg,    P =   -0.200 deg,    R =   -0.961 deg
};
P[639]{
   GP1:
    UF : 0, UT : 6,      CONFIG : 'N U T, 0, 0, 0',
    X =  350149.067  mm,    Y =   -50.934  mm,    Z =   -325826.947  mm,
    W =  -180.214 deg,    P =   -0.216 deg,    R =   -0.952 deg
};
P[640]{
   GP1:
    UF : 0, UT : 6,      CONFIG : 'N U T, 0, 0, 0',
    X =  349993.627  mm,    Y =   104.053  mm,    Z =   -325826.548  mm,
    W =  -179.930 deg,    P =   -0.263 deg,    R =   -0.962 deg
};
P[641]{
   GP1:
    UF : 0, UT : 6,      CONFIG : 'N U T, 0, 0, 0',
    X =  349982.826  mm,    Y =   114.408  mm,    Z =   -325826.150  mm,
    W =  -179.888 deg,    P =   -0.248 deg,    R =   -0.962 deg
};
P[642]{
   GP1:
    UF : 0, UT : 6,      CONFIG : 'N U T, 0, 0, 0',
    X =  350010.183  mm,    Y =   77.496  mm,    Z =   -325826.345  mm,
    W =  -180.024 deg,    P =   -0.172 deg,    R =   -0.985 deg
};
P[643]{
   GP1:
    UF : 0, UT : 6,      CONFIG : 'N U T, 0, 0, 0',
    X =  349916.816  mm,    Y =   130.140  mm,    Z =   -325826.365  mm,
    W =  -179.712 deg,    P =   -0.096 deg,    R =   -0.953 deg
};
P[644]{
   GP1:
    UF : 0, UT : 6,      CONFIG : 'N U T, 0, 0, 0',
    X =  349878.673  mm,    Y =   105.774  mm,    Z =   -325826.649  mm,
    W =  -179.695 deg,    P =   0.028 deg,    R =   -0.952 deg
};
P[645]{
   GP1:
    UF : 0, UT : 6,      CONFIG : 'N U T, 0, 0, 0',
    X =  350094.161  mm,    Y =   -118.362  mm,    Z =   -325826.129  mm,
    W =  -180.045 deg,    P =   0.031 deg,    R =   -0.998 deg
};
P[646]{
   GP1:
    UF : 0, UT : 6,      CONFIG : 'N U T, 0, 0, 0',
    X =  349868.486  mm,    Y =   92.821  mm,    Z =   -325826.685  mm,
    W =  -179.710 deg,    P =   0.060 deg,    R =   -0.955 deg
};
P[647]{
   GP1:
    UF : 0, UT : 6,      CONFIG : 'N U T, 0, 0, 0',
    X =  349983.300  mm,    Y =   -63.110  mm,    Z =   -325826.649  mm,
    W =  -179.922 deg,    P =   0.180 deg,    R =   -0.981 deg
};
P[648]{
   GP1:
    UF : 0, UT : 6,      CONFIG : 'N U T, 0, 0, 0',
    X =  349934.612  mm,    Y =   -15.316  mm,    Z =   -325826.682  mm,
    W =  -180.044 deg,    P =   0.187 deg,    R =   -0.981 deg
};
P[649]{
   GP1:
    UF : 0, UT : 6,      CONFIG : 'N U T, 0, 0, 0',
    X =  349858.729  mm,    Y =   60.859  mm,    Z =   -325826.873  mm,
    W =  -179.792 deg,    P =   0.135 deg,    R =   -0.969 deg
};
P[650]{
   GP1:
    UF : 0, UT : 6,      CONFIG : 'N U T, 0, 0, 0',
    X =  349974.774  mm,    Y =   -56.720  mm,    Z =   -325826.244  mm,
    W =  -179.947 deg,    P =   0.171 deg,    R =   -0.984 deg
};
P[651]{
   GP1:
    UF : 0, UT : 6,      CONFIG : 'N U T, 0, 0, 0',
    X =  349967.432  mm,    Y =   -51.345  mm,    Z =   -325826.266  mm,
    W =  -179.966 deg,    P =   0.157 deg,    R =   -0.987 deg
};
P[652]{
   GP1:
    UF : 0, UT : 6,      CONFIG : 'N U T, 0, 0, 0',
    X =  0.000  mm,    Y =   0.000  mm,    Z =   -225827.000  mm,
    W =  0.000 deg,    P =   0.000 deg,    R =   0.000 deg
};
/END
